Staubli VAL3: page_pallet.pjx

--- page_pallet.pjx ---
Parameters version=s7.7 stackSize=5000 millimeterUnit=true
Program file=buildList.pgx
Program file=insertInstr.pgx
Program file=listAdd.pgx
Program file=loadPage.pgx
Program file=main.pgx
Program file=onBackEvent.pgx
Program file=onEnterEvent.pgx
Program file=onExit.pgx
Program file=onF1Event.pgx
Program file=onF2Event.pgx
Program file=onF3Event.pgx
Program file=onF4Event.pgx
Program file=onF5Event.pgx
Program file=onF6Event.pgx
Program file=onF7Event.pgx
Program file=onF8Event.pgx
Program file=onStart.pgx
Program file=programList.pgx
Program file=refresh.pgx
Program file=refreshDynamic.pgx
Program file=refreshStatic.pgx
Program file=saveIt.pgx
Program file=setPallet.pgx
Data file=page_pallet.dtx
Library alias=page path=Disk://kernel/template/page/page.pjx
Library alias=use path=Disk://kernel/userPage/userPage.pjx
Library alias=language path=Disk://kernel/language/language.pjx
Library alias=saveData path=Disk://saveData/saveData.pjx
Library alias=pallet path=Disk://trajectory/PALLET/PALLET.pjx
Library alias=events path=Disk://..//templates/instruction/instruction.pjx
Library alias=prog path=Disk://instruction/PROG/PROG.pjx
Library alias=cycleStatus path=Disk://cycleStatus/cycleStatus.pjx
Library alias=language2 path=Disk://trajectory/PALLET/language/language.pjx
Library alias=tcp path=Disk://kernel/tool/tool.pjx
Type name=TrajPallet path=Disk://kernel/template/TrajPallet/TrajPallet.pjx
Type name=InstrItem path=Disk://kernel/template/InstrItem/InstrItem.pjx
Type name=FrameItem path=Disk://kernel/template/FrameItem/FrameItem.pjx

--- page_pallet.dtx ---
TrajPallet tTrajPallet
  [0]
    TrajPointItem tData
      [0]
        TrajectoryItem tSuper
          [0]
            num distance
            num moveType
            num nTime
            num nStop
            num nTcpAction
            string comment
            bool toStop
            mdesc nom_speed = {tmax=300, rmax=9999, leave=30, reach=30}
            InstrItem iInstr[3]
              [0]
                string sType
                string sData
              [1]
                string sType
                string sData
              [2]
                string sType
                string sData
            num nMoveId
        pointRx pPoint = {fatherId=tTrajPallet[0].fFrame[0]}
        num nType
    frame fFrame = {fatherId=tTrajPallet[0].fReference[0]}
    num nIndexTool
    string sID
    trsf trAppro[2]
      [0] = {z=-50}
      [1] = {z=-50}
    trsf trDepart[2]
      [0] = {z=-50}
      [1] = {z=-50}
    num nX = 1
    num nY = 1
    num nZ = 1
    num nIndex = 1
    num nDistanceXYZ[3]
      [0] = 1
      [1] = 1
      [2] = 1
    string sAction
    pointRx pO = {fatherId=tTrajPallet[0].fReference[0]}
    pointRx pX = {fatherId=tTrajPallet[0].fReference[0]}
    pointRx pY = {fatherId=tTrajPallet[0].fReference[0]}
    pointRx pZ = {fatherId=tTrajPallet[0].fReference[0]}
    num nSpeedApproach = 300
    num nSpeedDepart = 300
    num nIndexFrame
    frame fReference = {fatherId=world[0]}
bool bButton[8]
  [1] = true
  [4] = true
  [5] = true
  [6] = true
  [7] = true
bool bExit
bool bLarge
bool bOnActionLine
bool bToSave
num nIndex
num nKey = -1
num nPosition = 1
num nRefresh
num nTime = 2
pointRx pNull = {fatherId=world[0]}
pointRx pO = {fatherId=world[0]}
pointRx pOrigin = {fatherId=world[0]}
string sAction
string sEvent = "on Layer 1>"
public string sItems = "test"
string sList[8]
  [0] = "position > 2/1"
  [1] = "pos.  X  > 1/1"
  [2] = "pos.  Y  > 1/1"
  [3] = "pos.  Z  > 2/1"
  [4] = "  dX     > 1  "
  [5] = "  dY     > 1  "
  [6] = "  dZ     > 1  "
  [7] = "on Layer 1>"
string sMenu[8]
  [1] = "Edit Pallet"
  [4] = "Wizard"
  [5] = "Reset"
  [6] = "Back"
  [7] = "Next"
string sPalletName = "test"
num nView
frame fFather = {fatherId=world[0]}

--- main.pgx ---
public program main()
  local bool l_bSave
begin
  // INIT
  call onStart()
  // LOOP UNTIL nKey=255
  do
    call refresh()
    nKey=getKey()
    call use:listevent(nKey,nIndex,sEvent)
    nView=use:nView
    switch nKey
      case 259
        // TAB
        bLarge=!bLarge
        call use:setView(bLarge)
      break
      case 271
        // VIEW PROG
        call onF1Event(sAction)
      break
      case 272
        // edit traj
        call onF2Event(l_bSave)
      break
      case 273
        call onF3Event()
      break
      case 274
        call onF4Event()
      break
      case 275
        // wizard
        call onF5Event(l_bSave)
      break
      case 276
        // back
        call onF6Event(sPalletName)
      break
      case 277
        // next
        call onF7Event(sPalletName)
      break
      case 278
        // reset
        call onF8Event(sPalletName)
      break
      case 270
        call onEnterEvent(sPalletName,l_bSave)
      break
      case 263
        call onBackEvent(sPalletName,l_bSave)
      break
    endSwitch
    // look for the exit
    if nKey==255
      // on Exit
      call onExit(l_bSave)
    endIf
    // release
    delay(0)
  until bExit
  // reset the key pressure
  call use:nullKey(nKey)
end

--- buildList.pgx ---
program buildList()
  local num l_nSize
  local string l_sEvent
  local num i
  local num j
  local string l_sMessage
  local string l_sEmpty
  local TrajPallet l_tPallet
begin
  //
  // INIT the list
  l_sEmpty=""
  call use:stringCopy(l_sEmpty,sList)
  // Build the list
  call pallet:getSizeItem(false,l_nSize)
  call pallet:getPalletPos(sPalletName,nPosition)
  call pallet:getPalletData(false,l_tPallet)
  // show it
  call language2:message(l_sMessage,11)
  call use:strfill(l_sMessage,9,l_sMessage)
  call listAdd(l_sMessage+"> "+toString("",nPosition+1)+"/"+toString("",l_nSize))
  call language2:message(l_sMessage,12)
  call use:strfill(l_sMessage,9,l_sMessage)
  call listAdd(l_sMessage+"> "+toString("",(nPosition%(l_tPallet.nX*l_tPallet.nY))%l_tPallet.nX+1)+"/"+toString("",l_tPallet.nX))
  call language2:message(l_sMessage,13)
  call use:strfill(l_sMessage,9,l_sMessage)
  call listAdd(l_sMessage+"> "+toString("",roundDown((nPosition%(l_tPallet.nX*l_tPallet.nY))/l_tPallet.nX)+1)+"/"+toString("",l_tPallet.nY))
  call language2:message(l_sMessage,14)
  call use:strfill(l_sMessage,9,l_sMessage)
  call listAdd(l_sMessage+"> "+toString("",roundDown(nPosition/(l_tPallet.nX*l_tPallet.nY))+1)+"/"+toString("",l_tPallet.nZ))
  // show the x_y_z distance offset
  call listAdd("  dX     > "+toString(".1",l_tPallet.nDistanceXYZ[0]))
  call listAdd("  dY     > "+toString(".1",l_tPallet.nDistanceXYZ[1]))
  call listAdd("  dZ     > "+toString(".1",l_tPallet.nDistanceXYZ[2]))
  l_nSize=0
  for i=0 to size(l_tPallet.sAction)-1
    l_sEvent=l_tPallet.sAction[i]
    call language2:message(l_sMessage,15)
    call use:strfill(l_sMessage,9,l_sMessage)
    call listAdd(l_sMessage+toString("",i+1)+">"+l_sEvent)
  endFor
  // rebuild the list
  call use:listempty()
  call use:listadd(sList)
end

--- insertInstr.pgx ---
program insertInstr(InstrItem& x_sItem[])
  local num i
  local string l_sMessage
  local num l_nIndex
  local string l_sPath
  local string l_sItem
  local string l_sData
begin
  call use:setSizeList(19,0,19,11)
  call use:setView(false)
  call language2:message(l_sMessage,16)
  call use:listcreate(l_sMessage)
  // insert the action on Point
  call use:listadd(saveData:sInstrOnPoint)
  call use:listupdate(0)
  // SELECT THE ITEM
  x_sItem.sType=""
  x_sItem.sData=""
  do
    i=get()
    l_nIndex=0
    call use:listevent(i,l_nIndex,l_sItem)
  until i==255 or i==270
  //
  if l_sItem!="" and i==270
    call saveData:getPathInstr(l_sItem,l_sPath)
    events:libLoad(l_sPath)
    delay(0)
    call events:onInsert(l_sData)
    // insert the item
    x_sItem.sType=l_sItem
    x_sItem.sData=l_sData
    return
  endIf
  // NOT GOOD
  x_sItem.sType=""
  x_sItem.sData=""
  call use:nullKey(nKey)
end

--- listAdd.pgx ---
program listAdd(string x_sEvent (dimensions=1))
begin
  // add in the queue
  if sList!=""
    $dins(sList,size(sList))
  endIf
  sList[size(sList)-1]=x_sEvent
end

--- loadPage.pgx ---
program loadPage(string x_sPage, string& x_sItems[])
// load the next page
  local num i
  local string l_sMessage
begin
  // look if the page libload is correct
  i=page:libLoad(x_sPage)
  delay(0)
  if i!=0
    logMsg("[KERNEL] INTERFACE:PAGE LIBLOAD "+x_sPage+" result "+toString("",i))
    call language:message(l_sMessage,-7)
    popUpMsg(l_sMessage+x_sPage+" ; "+toString("",i))
  else
    // copy all the field from x_sItems to the next page
    call use:stringCopy(x_sItems,page:sItems)
    call page:main()
    // to give back
    call use:stringCopy(page:sItems,x_sItems)
  endIf
end

--- onBackEvent.pgx ---
program onBackEvent(string x_sName, bool& x_bSave[])
  local num i
  local string l_sProg
  local num l_nIndex
  local point l_pPoint[2]
  local string l_sEmpty
  local TrajPallet l_tPallet
  local num l_nPos
  local num l_nSize
  local num l_nXYZ[3]
  local num z
  local num y
  local num x
  local num l_nX
  local num l_nY
  local num l_nZ
  local num j
  local num l_nId
begin
  //
  // NB sEvent is the selected
  // element in the LIST
  //
  if nIndex>=0
    call use:findPos(sEvent,">",i)
    i=i+1
  endIf
  //
  // update all the value
  //
  call pallet:getSizeItem(false,l_nSize)
  call pallet:getPalletData(false,l_tPallet)
  call pallet:getPalletPos(x_sName,l_nPos)
  // make the default
  if l_nSize>=1
    // ORIGIN
    call pallet:getPoint(l_pPoint,false,0)
    fFather=tTrajPallet.fReference
    pO.trsf=position(l_pPoint,fFather)
    pOrigin.trsf=position(pO,l_tPallet.fFrame)
  endIf
  // clean the line
  call use:listcursor(use:nView,false)
  // swith the line
  // use this
  // l_nPos=(nX*nY)*(l_nZ-1)+(nX)*(l_nY-1)+(l_nX-1))
  // call setPalletPos(x_sItem,(l_nSize[0]*l_nSize[2])*(l_nValue[3]-1)+(l_nSize[0])*(l_nValue[2]-1)+(l_nValue[1]-1))
  l_nX=(l_nPos%(l_tPallet.nX*l_tPallet.nY))%l_tPallet.nX+1
  l_nY=roundDown((l_nPos%(l_tPallet.nX*l_tPallet.nY))/l_tPallet.nX)+1
  l_nZ=roundDown(l_nPos/(l_tPallet.nX*l_tPallet.nY))+1
  switch nIndex
    //
    default
      // plane line action
      if nIndex>=7
        l_tPallet.sAction[l_nIndex]=""
        x_bSave=true
      endIf
    break
  endSwitch
  // update the position
  if nIndex>=1 and nIndex<=3
    l_nPos=(l_tPallet.nX*l_tPallet.nY)*(l_nZ-1)+(l_tPallet.nX)*(l_nY-1)+(l_nX-1)
    call pallet:setPalletPos(x_sName,l_nPos)
  endIf
  // update all
  if x_bSave
    call pallet:setPalletData(l_tPallet)
    call pallet:getPalletData(false,tTrajPallet)
  endIf
  // refresh it
  call buildList()
  use:bUseRefresh=true
end

--- onEnterEvent.pgx ---
program onEnterEvent(string x_sName, bool& x_bSave[])
  local num i
  local string l_sProg
  local num l_nIndex
  local point l_pPoint[2]
  local string l_sEmpty
  local TrajPallet l_tPallet
  local num l_nPos
  local num l_nSize
  local num l_nXYZ[3]
  local num z
  local num y
  local num x
  local num l_nX
  local num l_nY
  local num l_nZ
  local num j
  local num l_nId
begin
  //
  // NB sEvent is the selected
  // element in the LIST
  //
  if nIndex>=0
    call use:findPos(sEvent,">",i)
    i=i+1
  endIf
  //
  // update all the value
  //
  call pallet:getSizeItem(false,l_nSize)
  call pallet:getPalletData(false,l_tPallet)
  call pallet:getPalletPos(x_sName,l_nPos)
  // make the default
  if l_nSize>=1
    // ORIGIN
    call pallet:getPoint(l_pPoint,false,0)

    fFather=tTrajPallet.fReference
    pO.trsf=position(l_pPoint,fFather)
    pOrigin.trsf=position(pO,l_tPallet.fFrame)
  endIf
  // clean the line
  call use:listcursor(use:nView,false)
  // swith the line
  // use this
  // l_nPos=(nX*nY)*(l_nZ-1)+(nX)*(l_nY-1)+(l_nX-1))
  // call setPalletPos(x_sItem,(l_nSize[0]*l_nSize[2])*(l_nValue[3]-1)+(l_nSize[0])*(l_nValue[2]-1)+(l_nValue[1]-1))
  l_nX=(l_nPos%(l_tPallet.nX*l_tPallet.nY))%l_tPallet.nX+1
  l_nY=roundDown((l_nPos%(l_tPallet.nX*l_tPallet.nY))/l_tPallet.nX)+1
  l_nZ=roundDown(l_nPos/(l_tPallet.nX*l_tPallet.nY))+1
  switch nIndex
    case 0
      // absolute
      l_sEmpty=""
      l_nPos=l_nPos+1
      call use:changeValue(l_nPos,1,l_nSize,i+40-use:nBottomX,use:nView+1,l_sEmpty)
      call pallet:setPalletPos(x_sName,l_nPos-1)
    break
    case 1
      // X value
      l_sEmpty=""
      call use:changeValue(l_nX,1,l_tPallet.nX,i+40-use:nBottomX,use:nView+1,l_sEmpty)
    break
    case 2
      // Y value
      l_sEmpty=""
      call use:changeValue(l_nY,1,l_tPallet.nY,i+40-use:nBottomX,use:nView+1,l_sEmpty)
    break
    case 3
      // Z value
      l_sEmpty=""
      call use:changeValue(l_nZ,1,l_tPallet.nZ,i+40-use:nBottomX,use:nView+1,l_sEmpty)
    break
    case 4,5,6
      // dx dy dz
      if l_nSize>1
        //get the old one
        for j=0 to 2
          l_nXYZ[j]=l_tPallet.nDistanceXYZ[j]
        endFor
        call use:changeValue(l_tPallet.nDistanceXYZ[nIndex-4],0,0,i+40-use:nBottomX,use:nView+1,l_sEmpty)
        // update it
        call pallet:setPalletData(l_tPallet)
        // set the offset
        l_nXYZ[0]=l_tPallet.nDistanceXYZ[0]-l_nXYZ[0]
        l_nXYZ[1]=l_tPallet.nDistanceXYZ[1]-l_nXYZ[1]
        l_nXYZ[2]=l_tPallet.nDistanceXYZ[2]-l_nXYZ[2]
        // change the offset for all
        call pallet:changeOffset(l_nXYZ)
        // update the value back
        call pallet:getPalletData(false,l_tPallet)
        use:bUseRefresh=true
        x_bSave=true
      endIf
    break
    //
    default
      // plane line action
      if nIndex>=7
        l_nIndex=nIndex-7
        l_sProg=right(sEvent,len(sEvent)-i)
        call programList(l_sProg)
        l_tPallet.sAction[l_nIndex]=l_sProg
        x_bSave=true
      endIf
    break
  endSwitch
  // update the position
  if nIndex>=1 and nIndex<=3
    l_nPos=(l_tPallet.nX*l_tPallet.nY)*(l_nZ-1)+(l_tPallet.nX)*(l_nY-1)+(l_nX-1)
    call pallet:setPalletPos(x_sName,l_nPos)
  endIf
  // update all
  if x_bSave
    call pallet:setPalletData(l_tPallet)
    call pallet:getPalletData(false,tTrajPallet)
  endIf
  // refresh it
  call buildList()
  use:bUseRefresh=true
end

--- onExit.pgx ---
program onExit(bool& x_bSave[] (dimensions=1))
  local string l_sMessage
  local bool l_bOk
  local string l_sButton[2]
  local bool l_bCancel
  local bool l_bYes
begin
  // saveIt
  if x_bSave
    call language:message(l_sMessage,-1)
    call language:getYesNo(l_sButton)
    // ask the yes_no question
    call use:yes_no_cancel(l_sMessage,l_sButton,l_bYes,l_bCancel)
    if l_bYes
      call saveIt(x_bSave)
    endIf
    // look for the cancel button
    bExit=!l_bCancel
  else
    // exit frome the page
    bExit=true
  endIf
end

--- onF1Event.pgx ---
program onF1Event(string x_sProg (dimensions=1))
  local string l_sPath
  local num l_nPath
begin
  // look if the bButton is enable
  if bButton[0]
    //
    // go to the edit program
    //
    l_sPath=prog:libPath()+"/page_viewInstr"
    call loadPage(l_sPath,x_sProg)
  endIf
end

--- onF2Event.pgx ---
program onF2Event(bool& x_bSave[] (dimensions=1))
  local string l_sPath
  local string l_sItems[2]
begin
  // look if the bButton is enable
  if bButton[1]
    //
    // edit all the pallet point
    //
    if x_bSave
      // saver IT
      call saveIt(x_bSave)
    endIf
    // load the page viewTraj
    l_sPath="Disk://trajectory/page_viewTraj"
    l_sItems=sPalletName
    nPosition=nPosition-1
    l_sItems[1]=toString("",max(nPosition[0],0))
    call loadPage(l_sPath,l_sItems)
    // came back
    if l_sItems[0]=="saved"
      x_bSave=false
    endIf
    //
    call buildList()
    //
  endIf
end

--- onF4Event.pgx ---
program onF4Event()
begin
  // look if the bButton is enable
  if bButton[3]
    //
  endIf
end

--- onF5Event.pgx ---
program onF5Event(bool& x_bSave[] (dimensions=1))
begin
  // look if the bButton is enable
  if bButton[4]
    //
    // Wizard
    call setPallet(x_bSave)
    // rebuild the list
    call buildList()
  endIf
end

--- onF6Event.pgx ---
program onF6Event(string x_sName (dimensions=1))
begin
  // look if the bButton is enable
  if bButton[5]
    // RESET
    call pallet:setPalletPos(x_sName,0)
    // refresh it
    call buildList()
    use:bUseRefresh=true
  endIf
end

--- onF7Event.pgx ---
program onF7Event(string x_sName (dimensions=1))
  local num l_nMax
begin
  // look if the bButton is enable
  if bButton[6]
    // BACK
    call pallet:back(x_sName)
    // refresh it
    call buildList()
    use:bUseRefresh=true
  endIf
end

--- onF8Event.pgx ---
program onF8Event(string x_sName (dimensions=1))
  local num l_nMax
begin
  // look if the bButton is enable
  if bButton[7]
    // NEXT
    call pallet:next(x_sName)
    // refresh it
    call buildList()
    use:bUseRefresh=true
  endIf
end

--- onStart.pgx ---
program onStart()
  local num i
  local string l_sPath
  local string l_sMessage
begin
  // logMsg
  logMsg("[KERNEL] INTERFACE:PAGE PALLET")
  // reset the exit button
  bExit=false
  // reset the Key pressure
  call use:nullKey(nKey)
  nIndex=0
  // load the TRAJ
  sPalletName=sItems
  // define the list
  call pallet:load(sPalletName,i)
  if i!=0
    call language:message(l_sMessage,-7)
    popUpMsg(l_sMessage+"#"+saveData:sTrajTypeUsing+"/"+sPalletName+" ; "+toString("",i))
  endIf
  //
  call buildList()
  // build the page
  call refreshStatic()
  // define the list
end

--- programList.pgx ---
program programList(string& x_sEvent[])
  local num nSize
  local string sEvent
  local num lKey
  local num i
  local string message
begin
  //
  // USE this procedure to view Prog
  // that you have already saved
  //
  cls()
  call use:setView(false)
  //
  // Prog
  //
  call use:listcreate("PROG ")
  // set the path to prog pallet
  //
  call prog:getSize(nSize)
  // refresh the list
  for i=0 to nSize-1
    call prog:get(sEvent,i)
    if sEvent!=""
      call use:listadd(sEvent)
    endIf
  endFor
  call use:listupdate(0)
  call language:message(message,60)
  call use:typeLen(0,13,message,40)
  call language:message(message,-19)
  message=" F7: "+message
  call use:type(0,9,message)
  do
    lKey=get()
    call use:listevent(lKey,i,x_sEvent)
  until lKey==270 or lKey==255 or lKey==277
  if lKey==277
    x_sEvent=""
  endIf
end

--- refreshDynamic.pgx ---
program refreshDynamic()
begin
  // DO NOT CHANGE
  nRefresh=clock()
  use:bUseRefresh=false
  //
  // ADD HERE
  //
  call buildList()
  //
  // refresh the cursor
  use:nView=nView
  // refresh the list
  call use:listupdate(nIndex-nView)
end

--- refreshStatic.pgx ---
program refreshStatic()
  local string l_sMenu
  local bool l_bOnActionLine
  local num l_nSize[4]
  local num i
  local num l_nIndex
  local TrajPallet l_tPallet
begin
  cls()
  //
  // set the view of the page..
  //
  // SET THE PAGE NUMBER
  use:nPage=10
  // USE <>PROFILE for <>PAGE
  use:nPage=use:nPage+abs(limit(saveData:mode,0,2)-2)
  if cycleStatus:bCycle
    use:nPage=use:nPage+3
  endIf
  // SET THE VIEW OF THE PAGE
  call language2:page(l_sMenu,use:nPage)
  //
  // define the menu
  call use:stringToArray(l_sMenu,sMenu)
  // enable/disabel the F1 Button
  l_bOnActionLine=false
  call pallet:getSizeItem(false,l_nSize)
  if nIndex>=0
    i=find(sEvent,">")+1
  endIf
  call pallet:getPalletData(false,l_tPallet)
//  if nIndex>=size(sList)-l_tPallet.nZ
//    //
//    l_nIndex=nIndex-size(sList)-l_tPallet.nZ
//    if l_tPallet.sAction[l_nIndex]!=""
//      l_bOnActionLine=true
//    endIf
//  endIf
  // set the menu
  if !bOnActionLine
    sMenu[0]=""
  endIf
  call use:setMenu(sMenu,true,3)
  call use:getMenu(sMenu,bButton)
  //
  // CREATE THE LIST
  //
  // define your list size for default
  call use:setSizeList(19,0,19,11)
  call use:setView(bLarge)
  //
  call use:listcreate("PALLET "+sPalletName)
  //
end

--- saveIt.pgx ---
program saveIt(bool& x_bSave[])
  local string l_sMessage
  local num l_nResult
  local string l_sEmpty
begin
  // save
  x_bSave=false
  logMsg("[KERNEL] INTERFACE:Save the trajectory "+saveData:sTrajTypeUsing+": "+sPalletName)
  call language:message(l_sMessage,-4)
  call use:timerDialog(l_sMessage,1)
  call pallet:setPalletData(tTrajPallet)
  call pallet:onSave(l_sEmpty)
end

--- setPallet.pgx ---
program setPallet(bool& x_bSave[])
  local string l_sMessage[3]
  local string l_sButton[8]
  local string l_sTcp
  local string l_sYesNo[2]
  local bool l_bDifferent
  local bool l_bCancel
  local num l_nStep
  local num l_nResult
  local num i
  local joint l_jPoint
  local point l_pPoint[2]
  local string l_sXYZline[3]
  local num l_nMin[3]
  local num l_nMax[3]
  local bool l_bRecompute
  local num l_nLineMin
  local num l_nLineMax
  local string l_sEmpty
  local num l_nApproach
  local bool l_bLinear
  local num l_nSpeed[3]
  local num l_nLine[3]
  local num l_nKey
  local num l_nIndex
  local num l_nDepart
  local num l_nSize
  local num x
  local num j
  local num z
  local num y
  local string l_sShow
  local string l_sSpeed
  local string l_sItem
  local num l_nId
begin
  //
  //  Change the Frame associate to the Pallet
  //
  //  take all the value
  //
  l_nStep=0
  l_sButton[0]=">>"
  l_sButton[1]="<<"
  call pallet:getTool(i)
  call tcp:getTool(saveData:tTool,i)
  saveData:nIndexTool=i
  call pallet:getPalletData(false,tTrajPallet)

  fFather=tTrajPallet.fReference
  // start it
  call language:message(l_sMessage,8)
  title("PALLET "+sPalletName+" "+l_sMessage)
  // WIZARD
  while l_nStep<10
    switch l_nStep
      case -1
        return
      break
      // select the TOOL
      // take the Origin-X-Y-Z
      case 0
        if !cycleStatus:bCycle
          cls()
          do
            call language:message(l_sMessage,150)
            call language:message(l_sMessage[1],167)
            call language:message(l_sMessage[2],190)
            call use:typeMenu(1,l_sMessage)
            call use:typeMenu(2,l_sMessage[1])
            call use:typeMenu(7,"<<")
            call use:typeMenu(8,">>")
            // show the here and the edit button
            call use:setSizeList(14,2,24,5)
            call use:listcreate(l_sMessage[2])
            // TOOL
            call language:message(l_sMessage,124)
            l_sItem=l_sMessage+": "+toString("3",saveData:nIndexTool)
            call use:listadd(l_sItem)
            //origin
            call language:message(l_sMessage,198)
            // pos. X
            call language2:message(l_sMessage[1],12)
            // pos. Y
            call language2:message(l_sMessage[2],13)
            call use:listadd(l_sMessage)
            // pos. Z
            call language2:message(l_sMessage[2],14)
            call use:listadd(l_sMessage[2])
            call use:listupdate(0)
            l_nKey=getKey()
            l_sEmpty=""
            call use:listevent(l_nKey,l_nResult,l_sEmpty)
            //
            if l_nResult!=l_nIndex or cycleStatus:nWorkingStatus!=0
              l_nIndex=l_nResult
              resetMotion()
            endIf
            switch l_nResult
              case 0
                if l_nKey==270
                  // TOOL
                  l_sEmpty=""
                  call loadPage("Disk://kernel/page/tool",l_sEmpty)
                  call tcp:getTool(saveData:tTool,saveData:nIndexTool)
                  tTrajPallet.nIndexTool=saveData:nIndexTool
                  // release
                  call use:nullKey(l_nKey)
                  cls()
                endIf
              break
              case 1
                // take the Origin
                if pointToJoint(saveData:tTool,herej(),tTrajPallet.pO,l_jPoint) and cycleStatus:nWorkingMode==1 and isEmpty()
                  movej(tTrajPallet.pO,saveData:tTool,{25,25,25,9999,9999,off,50,50})
                endIf
                //
                if l_nKey==271
                  tTrajPallet.pO=here(saveData:tTool,fFather)
                  l_sMessage=" [x] "
                  call use:type(2,4,l_sMessage)
                  // compute the point again
                  l_bRecompute=true
                elseIf l_nKey==272 or l_nKey==270
                  call language:message(l_sMessage,198)
                  call use:changeTrsf(tTrajPallet.pO.trsf,l_sMessage,"")
                  // compute the point again
                  l_bRecompute=true
                  cls()
                endIf
              break
              case 2
                //take the X Point
                if pointToJoint(saveData:tTool,herej(),tTrajPallet.pX,l_jPoint) and cycleStatus:nWorkingMode==1 and isEmpty()
                  movej(tTrajPallet.pX,saveData:tTool,{25,25,25,9999,9999,off,50,50})
                endIf
                // key pressure
                if l_nKey==271
                  tTrajPallet.pX=here(saveData:tTool,fFather)
                  l_sMessage=" [x] "
                  call use:type(2,5,l_sMessage)
                  // compute the point again
                  l_bRecompute=true
                elseIf l_nKey==272 or l_nKey==270
                  call language:message(l_sMessage,199)
                  call use:changeTrsf(tTrajPallet.pX.trsf,l_sMessage+" X","")
                  // compute the point again
                  l_bRecompute=true
                  cls()
                endIf
              break
              case 3
                // take the Y Point
                if pointToJoint(saveData:tTool,herej(),tTrajPallet.pY,l_jPoint) and cycleStatus:nWorkingMode==1 and isEmpty()
                  movej(tTrajPallet.pY,saveData:tTool,{25,25,25,9999,9999,off,50,50})
                endIf
                // key pressure
                if l_nKey==271
                  tTrajPallet.pY=here(saveData:tTool,fFather)
                  l_sMessage=" [x] "
                  call use:type(2,6,l_sMessage)
                  // compute the point again
                  l_bRecompute=true
                elseIf l_nKey==272 or l_nKey==270
                  call language:message(l_sMessage,199)
                  call use:changeTrsf(tTrajPallet.pY.trsf,l_sMessage+" Y","")
                  // compute the point again
                  l_bRecompute=true
                  cls()
                endIf
              break
              case 4
                // take the Z point
                if pointToJoint(saveData:tTool,herej(),tTrajPallet.pZ,l_jPoint) and cycleStatus:nWorkingMode==1 and isEmpty()
                  movej(tTrajPallet.pZ,saveData:tTool,{25,25,25,9999,9999,off,50,50})
                endIf
                // key pressure
                if l_nKey==271
                  tTrajPallet.pZ=here(saveData:tTool,fFather)
                  l_sMessage=" [x] "
                  call use:type(2,7,l_sMessage)
                  // compute the point again
                  l_bRecompute=true
                else
                  if l_nKey==272 or l_nKey==270
                    call language:message(l_sMessage,199)
                    call use:changeTrsf(tTrajPallet.pZ.trsf,l_sMessage+" Z","")
                    // compute the point again
                    l_bRecompute=true
                    cls()
                  else
                    call use:clear(0,11)
                  endIf
                endIf
              break
            endSwitch
            use:nView=l_nResult
            delay(0)
          until l_nKey==278 or l_nKey==277 or l_nKey==255 or l_nKey==264 or l_nKey==268
          // validate
          switch l_nKey
            case 278,268
              l_nResult=0
            break
            case 277,264
              l_nResult=2
            break
            case 255
              l_nResult=-1
            break
          endSwitch
          //
          // check the point[2] if point[1]
          //
          if l_nResult!=-1
            if tTrajPallet.pX.trsf!=tTrajPallet.pY.trsf and tTrajPallet.pO.trsf!=tTrajPallet.pY.trsf and tTrajPallet.pY.trsf!={0,0,0,0,0,0}
              // set the frame
              if setFrame(tTrajPallet.pO,tTrajPallet.pX,tTrajPallet.pY,tTrajPallet.fFrame)!=0
                // if not put a message
                call language2:message(l_sMessage,32)
                popUpMsg(l_sMessage)
                // came back
                l_nResult=2
              endIf
            elseIf tTrajPallet.pO.trsf!=tTrajPallet.pX.trsf and tTrajPallet.pO.trsf!={0,0,0,0,0,0}
              // try to put the y to fFather with the same Z as the origin point
              l_pPoint=here(saveData:tTool,fFather)
              l_pPoint.trsf=position(tTrajPallet.pO,fFather)
              l_pPoint.trsf={0,0,l_pPoint.trsf.z,0,0,0}
              if setFrame(tTrajPallet.pO,tTrajPallet.pX,l_pPoint,tTrajPallet.fFrame)!=0
                // if not put a message
                call language2:message(l_sMessage,32)
                popUpMsg(l_sMessage)
                // came back
                l_nResult=2
              endIf
            endIf
          endIf
        endIf
      break
      // set the OPTION
      case 1
        l_nResult=100
        do
          // BUILD THE LIST
          call language:message(l_sMessage,167)
          l_sButton[0]=">>"
          l_sButton[1]="<<"
          l_sButton[2]=""
          l_sButton[3]=""
          l_sButton[4]=""
          l_sButton[5]=""
          l_sButton[6]=l_sMessage
          l_sButton[7]=""
          call use:typeMenu(7,"<<")
          call use:typeMenu(8,">>")
          call use:typeMenu(2,l_sMessage)
          // create the list
          call use:setSizeList(16,2,22,6)
          call language:message(l_sItem,167)
          call use:listcreate(l_sItem)
          // take how many X,Y,Z lines
          l_nLine[0]=tTrajPallet.nX
          l_nLine[1]=tTrajPallet.nY
          l_nLine[2]=tTrajPallet.nZ
          l_sItem="Line: "+toString("",tTrajPallet.nX)+","+toString("",tTrajPallet.nY)+","+toString("",tTrajPallet.nZ)
          call use:listadd(l_sItem)
          call language2:message(l_sItem,3)
          l_sItem=l_sItem+": "+toString("",-tTrajPallet.trAppro.z)
          call use:listadd(l_sItem)
          call language2:message(l_sItem,4)
          l_sItem=l_sItem+": "+toString("",-tTrajPallet.trDepart.z)
          call use:listadd(l_sItem)
          // linear move or not
          call language:message(l_sMessage,157)
          call language:message(l_sMessage[1],164+tTrajPallet.tData.tSuper.moveType)
          l_sItem=l_sMessage+":"+l_sMessage[1]
          l_bLinear=tTrajPallet.tData.tSuper.moveType==1
          call use:listadd(l_sItem)
          // show the speed
          call language:message(l_sSpeed,158)
          l_sSpeed=l_sSpeed+": "+toString("",tTrajPallet.nSpeedApproach)+","
          l_sSpeed=l_sSpeed+toString("",tTrajPallet.nSpeedDepart)+","
          if !l_bLinear
            // JOINT Move
            l_sSpeed=l_sSpeed+toString("",tTrajPallet.tData.tSuper.nom_speed.vel)+"%"
          else
            // Linear Move
            l_sSpeed=l_sSpeed+toString("",tTrajPallet.tData.tSuper.nom_speed.tvel)+"mm/sec"
          endIf
          call use:listadd(l_sSpeed)
          // STOP time
          call language:message(l_sMessage,174)
          l_sItem=l_sMessage+": "+toString(".2",tTrajPallet.tData.tSuper.nStop)
          call use:listadd(l_sItem)
          // update it
          call use:listupdate(0)
          l_nKey=get()
          call use:listevent(l_nKey,l_nIndex,l_sMessage)
          // key event
          if l_nKey==270 or l_nKey==32 or l_nKey==272
            switch l_nIndex
              case 0
                cls()
                l_sButton[7]=""
                l_sButton[6]=""
                // set the message
                //line X
                call language2:message(l_sMessage,18)
                l_sXYZline[0]=l_sMessage
                // line Y
                if tTrajPallet.pY.trsf!={0,0,0,0,0,0}
                  call language2:message(l_sMessage,19)
                  l_sXYZline[1]=l_sMessage
                endIf
                // line Z
                if tTrajPallet.pZ.trsf!={0,0,0,0,0,0}
                  call language2:message(l_sMessage,20)
                  l_sXYZline[2]=l_sMessage
                endIf
                l_nLineMin=0
                l_nLineMax=100
                call use:editNumField("PALLET X Y Z",l_sXYZline,l_nLine,l_nLineMin,l_nLineMax)
                // check the size
                l_bDifferent=false
                if l_nLine[0]!=tTrajPallet.nX or l_nLine[1]!=tTrajPallet.nY or l_nLine[2]!=tTrajPallet.nZ
                  l_bDifferent=true
                  tTrajPallet.nX=l_nLine[0]
                  tTrajPallet.nY=l_nLine[1]
                  tTrajPallet.nZ=l_nLine[2]
                else
                  l_bDifferent=false
                endIf
              break
              case 1
                // APPROACH
                call language:message(l_sMessage,167)
                call use:typeMenu(2,l_sMessage)
                // look for the approach
                if tTrajPallet.trAppro[0]==tTrajPallet.trAppro[1] and (tTrajPallet.trAppro.x==0 and tTrajPallet.trAppro.y==0 and tTrajPallet.trAppro.rx==0 and tTrajPallet.trAppro.ry==0 and tTrajPallet.trAppro.rz==0) and l_nKey==270
                  // normal Approach only Z
                  call language2:message(l_sMessage,21)
                  l_nApproach=-tTrajPallet.trAppro.z
                  call use:insertDialog(l_sMessage,l_nApproach,0,999)
                  tTrajPallet.trAppro=tTrajPallet.trAppro[1]={0,0,-l_nApproach,0,0,0}
                  // edit IT
                else
                  // TRSF APPROACH
                  call language2:message(l_sMessage,40)
                  call language2:message(l_sMessage[1],42)
                  if tTrajPallet.trAppro==tTrajPallet.trAppro[1] and tTrajPallet.trAppro=={0,0,0,0,0,0}
                    // change the approach 1
                    call use:changeTrsf(tTrajPallet.trAppro,l_sMessage+" [1]",l_sMessage[1])
                    tTrajPallet.trAppro[1]=tTrajPallet.trAppro
                  else
                    call use:changeTrsf(tTrajPallet.trAppro,l_sMessage+" [1]",l_sMessage[1])
                  endIf
                  // change the approach 2
                  call use:changeTrsf(tTrajPallet.trAppro[1],l_sMessage+" [2]",l_sMessage[1])
                endIf
              break
              case 2
                // DEPART
                call language:message(l_sMessage,167)
                call use:typeMenu(2,l_sMessage)
                // look for the depart
                if tTrajPallet.trDepart==tTrajPallet.trDepart[1] and (tTrajPallet.trDepart.x==0 and tTrajPallet.trDepart.y==0 and tTrajPallet.trDepart.rx==0 and tTrajPallet.trDepart.ry==0 and tTrajPallet.trDepart.rz==0) and l_nKey==270
                  // normal Depart only Z
                  l_nDepart=-tTrajPallet.trDepart.z
                  call language2:message(l_sMessage,22)
                  call use:insertDialog(l_sMessage,l_nDepart,0,999)
                  tTrajPallet.trDepart=tTrajPallet.trDepart[1]={0,0,-l_nDepart,0,0,0}
                else
                  // TRSF DEPART
                  call language2:message(l_sMessage,41)
                  call language2:message(l_sMessage[1],42)
                  if tTrajPallet.trDepart==tTrajPallet.trDepart[1] and tTrajPallet.trDepart=={0,0,0,0,0,0}
                    // change the approach 1
                    call use:changeTrsf(tTrajPallet.trDepart,l_sMessage+" [1]",l_sMessage[1])
                    tTrajPallet.trDepart[1]=tTrajPallet.trDepart
                  else
                    call use:changeTrsf(tTrajPallet.trDepart,l_sMessage+" [1]",l_sMessage[1])
                  endIf
                  // change the approach 2
                  call use:changeTrsf(tTrajPallet.trDepart[1],l_sMessage+" [2]",l_sMessage[1])
                endIf
              break
              case 3
                if l_nKey==270 or l_nKey==32
                  l_bLinear=!l_bLinear
                  tTrajPallet.tData.tSuper.moveType=sel(l_bLinear,1,0)
                  // check the moveType
                  if tTrajPallet.tData.tSuper.moveType==1
                    // convert to LINEAR
                    tTrajPallet.tData.tSuper.nom_speed.tvel=600
                    tTrajPallet.tData.tSuper.nom_speed.vel=450
                  elseIf tTrajPallet.tData.tSuper.moveType==0
                    // convert TO JOINT
                    tTrajPallet.tData.tSuper.nom_speed.tvel=9999
                    tTrajPallet.tData.tSuper.nom_speed.vel=50
                  endIf
                endIf
              break
              case 4
                if l_nKey==270 or l_nKey==32
                  // go to the default
                  call language:message(l_sMessage[2],158)
                  // take the speed approach
                  l_nSpeed[0]=tTrajPallet.nSpeedApproach
                  call language2:message(l_sMessage[0],40)
                  l_sMessage[0]=l_sMessage[0]+" "+l_sMessage[2]+" mm/sec"
                  l_nMin[0]=1
                  l_nMax[0]=2000
                  // take the speed Depart
                  l_nSpeed[1]=tTrajPallet.nSpeedDepart
                  call language2:message(l_sMessage[1],41)
                  l_sMessage[1]=l_sMessage[1]+" "+l_sMessage[2]+" mm/sec"
                  l_nMin[1]=1
                  l_nMax[1]=2000
                  // take the speed
                  if tTrajPallet.tData.tSuper.moveType==0
                    call language:message(l_sMessage[2],158)
                    l_sMessage[2]=l_sMessage[2]+" % "
                    l_nSpeed[2]=tTrajPallet.tData.tSuper.nom_speed.vel
                    l_nMin[2]=10
                    l_nMax[2]=200
                  else
                    call language:message(l_sMessage[2],158)
                    l_sMessage[2]=l_sMessage[2]+" mm/sec"
                    l_nSpeed[2]=tTrajPallet.tData.tSuper.nom_speed.tvel
                    l_nMin[2]=100
                    l_nMax[2]=20000
                  endIf
                  // edit the field
                  call use:editNumField("",l_sMessage,l_nSpeed,l_nMin,l_nMax)
                  // copy back
                  tTrajPallet.nSpeedApproach=l_nSpeed[0]
                  tTrajPallet.nSpeedDepart=l_nSpeed[1]
                  if  tTrajPallet.tData.tSuper.moveType==0
                    tTrajPallet.tData.tSuper.nom_speed.vel=l_nSpeed[2]
                    tTrajPallet.tData.tSuper.nom_speed.tvel=9999
                  else
                    tTrajPallet.tData.tSuper.nom_speed.tvel=l_nSpeed[2]
                    tTrajPallet.tData.tSuper.nom_speed.vel=450
                  endIf
                endIf
              break
              case 5
                if l_nKey==270 or l_nKey==32
                  // STOP TIME
                  call language2:message(l_sMessage,43)
                  call use:insertDialog(l_sMessage,tTrajPallet.tData.tSuper.nStop,0,10)
                endIf
              break
            endSwitch
            // release
            call use:nullKey(l_nKey)
            cls()
          elseIf l_nKey==278 or l_nKey==268
            l_nResult=0
          elseIf l_nKey==277 or l_nKey==264
            l_nResult=2
          elseIf l_nKey==255
            l_nResult=-1
          endIf
          //
          // release
          delay(0)
        until l_nResult!=100
      break
      case 2
        // take the instruction
        //  Insert the first instruction
        //
        l_sButton[0]=">>>"
        l_sButton[1]="<<"
        l_sButton[2]=""
        l_sButton[3]=""
        l_sButton[4]=""
        l_sButton[5]="NONE"
        l_sButton[6]="ON"
        l_sButton[5]="OFF"
        l_sButton[7]="INSTR"
        if tTrajPallet.tData.tSuper.nTcpAction==1
          l_sMessage="ON "
        elseIf tTrajPallet.tData.tSuper.nTcpAction==2
          l_sMessage="OFF"
        else
          l_sMessage="..."
        endIf
        call use:type(2,10,"TCP-> "+l_sMessage)
        call language2:message(l_sMessage,26)
        call use:questionDialog(l_sMessage,l_sButton,l_nResult)
        switch l_nResult
          case 8
            call insertInstr(tTrajPallet.tData[0].tSuper.iInstr)
          break
          case 7
            // SET TCP ON
            tTrajPallet.tData.tSuper.nTcpAction=1
          break
          case 6
            // SET TCP OFF
            tTrajPallet.tData.tSuper.nTcpAction=2
          break
          case 5
            // empty all
            tTrajPallet.tData.tSuper.nTcpAction=0
            tTrajPallet.tData[0].tSuper.iInstr.sType=""
            tTrajPallet.tData[0].tSuper.iInstr.sData=""
          break
          case 0,1
            // go to end
          break
        endSwitch
      break
      case 3
        // REBUILD the pallet
        l_sButton[7]=""
        l_nSize=l_nLine[0]*l_nLine[1]*l_nLine[2]
        // calcolate the distance
        if l_bDifferent or l_bRecompute
          // POINT X
          if l_nLine[0]>1
            l_pPoint=here(flange,tTrajPallet.fFrame)
            l_pPoint.trsf=position(tTrajPallet.pX,tTrajPallet.fFrame)
             tTrajPallet.nDistanceXYZ[0]=l_pPoint.trsf.x/(l_nLine-1)
          else
            tTrajPallet.nDistanceXYZ[0]=0
          endIf
          // POINT Y
          if l_nLine[1]>1
            l_pPoint=here(flange,tTrajPallet.fFrame)
            l_pPoint.trsf=position(tTrajPallet.pY,tTrajPallet.fFrame)
            tTrajPallet.nDistanceXYZ[1]=abs(l_pPoint.trsf.y/(l_nLine[1]-1))
          else
            tTrajPallet.nDistanceXYZ[1]=0
          endIf
          // POINT Z
          if l_nLine[2]>1
            // put the point Z in the tTrajPallet.fFrame frame to have the good distance
            l_pPoint=here(flange,tTrajPallet.fFrame)
            l_pPoint.trsf=position(tTrajPallet.pZ,tTrajPallet.fFrame)
            tTrajPallet.nDistanceXYZ[2]=l_pPoint.trsf.z/(l_nLine[2]-1)
          else
            tTrajPallet.nDistanceXYZ[2]=0
          endIf
          // calcolate all the point
          link(pOrigin,tTrajPallet.fFrame)
          pOrigin.trsf=position(tTrajPallet.pO,tTrajPallet.fFrame)
          // Redifine the size
          if l_bDifferent
            resize(tTrajPallet.tData,1,l_nSize)
            resize(tTrajPallet.sAction,1,l_nLine[2])
          endIf
          // save the change...
          i=0
          l_bCancel=false
          for z=0 to tTrajPallet.nZ-1
            for y=0 to tTrajPallet.nY-1
              for x=0 to tTrajPallet.nX-1
                l_pPoint=compose(pOrigin,tTrajPallet.fFrame,{tTrajPallet.nDistanceXYZ[0]*x,tTrajPallet.nDistanceXYZ[1]*y,tTrajPallet.nDistanceXYZ[2]*z,0,0,0})
                // check the point config
                // set the data
                tTrajPallet.tData[i].pPoint.trsf=l_pPoint.trsf
                link(tTrajPallet.tData[i].pPoint,tTrajPallet.fFrame)
                tTrajPallet.tData[i].tSuper.comment="("+toString("",x+1)+","+toString("",y+1)+","+toString("",z+1)+")"
                // increase the index
                i=i+1
                if !pointToJoint(saveData:tTool,herej(),l_pPoint,l_jPoint)
                  l_bCancel=true
                  popUpMsg("the point: "+toString("",i)+" is not accessible...")
                endIf
              endFor
            endFor
          endFor
        endIf
        for i=0 to l_nSize-1
          // copy all the value from the first element
          tTrajPallet.tData[i].tSuper.moveType=tTrajPallet.tData[0].tSuper.moveType
          tTrajPallet.tData[i].tSuper.nStop=tTrajPallet.tData[0].tSuper.nStop
          tTrajPallet.tData[i].tSuper.nTcpAction=tTrajPallet.tData[0].tSuper.nTcpAction
          tTrajPallet.tData[i].tSuper.toStop=tTrajPallet.tData[0].tSuper.toStop
          tTrajPallet.tData[i].tSuper.nom_speed=tTrajPallet.tData[0].tSuper.nom_speed
          for j=0 to size(tTrajPallet.tData[i].tSuper.iInstr[j])-1
            tTrajPallet.tData[i].tSuper.iInstr[j].sType=tTrajPallet.tData[0].tSuper.iInstr[j].sType
            tTrajPallet.tData[i].tSuper.iInstr[j].sData=tTrajPallet.tData[0].tSuper.iInstr[j].sData
          endFor
        endFor
        //
        // save
        //
        tTrajPallet.fReference.trsf=saveData:fFrameItem[tTrajPallet.nIndexFrame].fFrame.trsf
        call pallet:setPalletData(tTrajPallet)
        x_bSave=true
        // check
        if !l_bCancel
          popUpMsg("Pallet OK")
        endIf
        return
      break
      //
    endSwitch
    // release
    call use:nullKey(l_nKey)
    // step control
    if l_nResult==0 or l_nResult==1
      l_nStep=l_nStep+1
      // clear the screen
      cls()
    else
      if l_nResult==2
        l_nStep=l_nStep-1
        // clear the screen
        cls()
      else
        if l_nResult==-1
          // check if the pallet already exist
          if l_nLine>=1
            // ask if they want to save the config
            call language2:message(l_sMessage,31)
            // get the yes_no button
            call language:getYesNo(l_sYesNo)
            // ask the question
            call use:yes_no_cancel(l_sMessage,l_sYesNo,l_bDifferent,l_bCancel)
            if !l_bCancel
              if l_bDifferent
                // save the last modification
                l_nStep=3
              else
                // exit
                return
              endIf
            endIf
          else
            // exit without saving
            return
          endIf
        endIf
      endIf
    endIf
  endWhile
end
